{attribute 'qualified_only'}
VAR_GLOBAL
	fbMyNewConfiguration		: FB_MyNewConfiguration;
	
END_VAR

(* stored: Version 1.1.0.1, ProductVersion 3.1.4024.15
   GVL GVL_Variable: Id {6a962dfd-5722-4359-8bb2-411af6f813c5} *)
